// TIA Portal V19 export
TYPE "LPMLV2022_typeDiagnosticsEntry"
TITLE = LPMLV2022_typeDiagnosticsEntry
// Support: tech.team.motioncontrol@siemens.com
// stored: Access Published
   STRUCT
      timestamp { ExternalWritable := 'False'} : DTL;   // Timestamp for this entry
      UnitModeCurrent { ExternalWritable := 'False'} : SInt;   // Current unit mode
      StateCurrent { ExternalWritable := 'False'} : SInt;   // Current state
      UnitMode { ExternalWritable := 'False'} : SInt;   // Requested unit mode
      CntrlCmd { ExternalWritable := 'False'} : SInt;   // Request control command
      SC { ExternalWritable := 'False'} : Bool;   // State complete signal
      message { ExternalWritable := 'False'} : Byte;   // Message for this entry
   END_STRUCT;
END_TYPE
